TYPE EL922x_ChannelExtended :
STRUCT
	Status AT%I* : StatusStructExtended;
	Load AT%I* : UINT;
	Current AT%I* : UINT;
	VoltageIn AT%I* : UINT;
	VoltageOut AT%I* : UINT;
	Control AT%q* : OutputStruct;
END_STRUCT
END_TYPE

(* stored: Version 1.1.0.1, ProductVersion 3.1.4024.5
   DUT EL922x_ChannelExtended: Id {6d74edf6-7f49-4973-820c-49d572e4802a} *)
